INTERFACE ITF_Schuif_AnaIn_AFO

METHOD get : SINT
VAR_INPUT
END_VAR
END_METHOD

END_INTERFACE

(* stored: Version 1.1.0.1, ProductVersion 3.1.4026.8
   Itf ITF_Schuif_AnaIn_AFO: Id {ff3ed898-1395-46ff-8850-405f840f374d}
   Method get: Id {c473f6ef-f3e0-400c-baa7-85fae2eaa728} *)
